// TIA Portal V19 export
TYPE "LubrMotor_Par"
// stored: Access Published
   STRUCT
      EnableCheckRotation : Bool;   // Enable check the motor rotation feedback
      LowLevelCheckTime : Time;
      RotationFbkCheckTime : Time;   // Time to check the motor rotation feedback
   END_STRUCT;
END_TYPE
